(* CODESYS project Library.library
   Company: HDS Global
   Title: RoboFS_Standard
   Placeholder: RoboFS_Standard
   Version: 1.0

Project tree, tasks and I/O mapping:
  libraries: Tc2_MC2, * (Beckhoff Automation GmbH); Tc2_Standard, * (Beckhoff Automation GmbH); Tc2_System, * (Beckhoff Automation GmbH); Tc3_Module, * (Beckhoff Automation GmbH)
  Assemblies/
    function block Assembly_Conveyor [ST]
    function block Assembly_LAT [ST]
    function block Assembly_Lift [ST]
  Device Controllers/
    function block Device_Actuator [ST]
    function block Device_Motor_OnOff [ST]
    function block Device_PartSensor [FBD]
    function block Device_Servo [ST]: Disabled, Disabling, Enabled, Enabling, Error, Homing, Jogging, MoveComplete, MoveInProgress, Resetting, Stopped, Stopping
  DUTs/
    data type eInput
    data type Handshake_Receive
    data type Handshake_Send
    data type Intfc_Receiver
    data type Intfc_Sender
    data type ServoMove
  Enumerations/
    data type Cmd
    data type CmdActuator
    data type CmdMotorOnOff
    data type CmdServo
    data type Mode
    data type MoveTypeServo
    data type State
    data type StateActuator
    data type StateMotorOnOff
    data type StateSequencer
    data type StateServo
    data type StatusStep
  Instructions/
    function block eAND [ST]
    function block eOR [ST]
    function block MC_MoveParametersCheck [ST]
    function block StateManager [ST]
    function block Step [ST]
  Version/
    global variables Global_Version
*)

// DUTs/eInput
TYPE eInput :
STRUCT
	iState			: BOOL;
	iForceActive 	: BOOL;
	iForceInactive	: BOOL;
	cName			: STRING;
	cActiveState 	: BOOL := TRUE;
	oActive			: BOOL;
END_STRUCT
END_TYPE

// DUTs/Handshake_Receive
TYPE Handshake_Receive :
STRUCT
	ReadyToReceive 	: BOOL;
	Received		: BOOL;
	PartInfo		: STRING(20);
END_STRUCT
END_TYPE

// DUTs/Handshake_Send
TYPE Handshake_Send :
STRUCT
	WaitingToSend	: BOOL;
	Sending			: BOOL;
	PartInfo		: STRING(20);
END_STRUCT
END_TYPE

// DUTs/Intfc_Receiver
TYPE Intfc_Receiver :
STRUCT
	iHandshake 			: Handshake_Send;
	oHandshake			: Handshake_Receive;
	cSenderNetId		: STRING;
	cSenderPort			: UINT;
END_STRUCT
END_TYPE

// DUTs/Intfc_Sender
TYPE Intfc_Sender :
STRUCT
	oHandshake				: Handshake_Send;
	iHandshake		 		: Handshake_Receive;
	cReceiverNetId			: STRING;
	cReceiverPort			: UINT;
END_STRUCT
END_TYPE

// DUTs/ServoMove
TYPE ServoMove :
STRUCT
	Name 		: STRING;
	MoveType	: MoveTypeServo;
	Position	: LREAL;
	Velocity	: LREAL;
	Accel		: LREAL;
	Decel		: LREAL;
	Jerk		: LREAL;
	Direction	: MC_Direction;
	BufferMode	: MC_BufferMode;
	Permissive	: eAND;
	Interlock	: eAND;
END_STRUCT
END_TYPE

// Enumerations/Cmd
{attribute 'qualified_only'}
{attribute 'strict'}
TYPE Cmd :
(
	None,
	Abort,
	Reset,
	Start,
	Stop,
	Pause,
	Resume
);
END_TYPE

// Enumerations/CmdActuator
{attribute 'qualified_only'}
{attribute 'strict'}
TYPE CmdActuator :
(
	None,
	Extend,
	Retract,
	Reset
);
END_TYPE

// Enumerations/CmdMotorOnOff
{attribute 'qualified_only'}
{attribute 'strict'}
TYPE CmdMotorOnOff :
(
	None,
	Reset,
	StartFwd,
	StartRev,
	Stop	
);
END_TYPE

// Enumerations/CmdServo
{attribute 'qualified_only'}
{attribute 'strict'}
TYPE CmdServo :
(
	None,
	Enable,
	Disable,
	Reset,
	Home,
	StartMove,
	Stop,
	Jog
);
END_TYPE

// Enumerations/Mode
{attribute 'qualified_only'}
{attribute 'strict'}
TYPE Mode :
(
	Auto,
	Manual
);
END_TYPE

// Enumerations/MoveTypeServo
{attribute 'qualified_only'}
{attribute 'strict'}
TYPE MoveTypeServo :
(
	None,
	Continuous,
	LinearAbs,
	LinearRel,
	RotaryAbs,
	RotaryRel
);
END_TYPE

// Enumerations/State
{attribute 'qualified_only'}
{attribute 'strict'}
TYPE State :
(
	None,
	Stopped,
	Starting,
	Running,
	Pausing,
	Paused,
	Resuming,
	Stopping,
	Aborting,
	Aborted,
	Resetting	
);
END_TYPE

// Enumerations/StateActuator
{attribute 'qualified_only'}
{attribute 'strict'}
TYPE StateActuator :
(
	None,
	Error,
	Retracting,
	Retracted,
	Extending,
	Extended
);
END_TYPE

// Enumerations/StateMotorOnOff
{attribute 'qualified_only'}
{attribute 'strict'}
TYPE StateMotorOnOff :
(
	None,
	Error,
	Stopping,
	Stopped,
	StartingFwd,
	RunningFwd,
	StartingRev,
	RunningRev
);
END_TYPE

// Enumerations/StateSequencer
{attribute 'qualified_only'}
{attribute 'strict'}
TYPE StateSequencer :
(
	Idle,
	Running,
	Complete,
	Faulted
);
END_TYPE

// Enumerations/StateServo
{attribute 'qualified_only'}
{attribute 'strict'}
TYPE StateServo :
(
	None,
	Error,
	Resetting,
	Disabling,
	Disabled,
	Enabling,
	Enabled,
	Homing,
	MoveInProgress,
	MoveComplete,
	Stopping,	
	Stopped,
	Jogging
);
END_TYPE

// Enumerations/StatusStep
{attribute 'qualified_only'}
{attribute 'strict'}
TYPE StatusStep :
(
	Inactive,
	Active,
	Faulted,
	TimedOut,
	Complete
);
END_TYPE

// Version/Global_Version
{attribute 'TcGenerated'}
// This function has been automatically generated from the project information.
VAR_GLOBAL CONSTANT
	{attribute 'const_non_replaced'}
	{attribute 'linkalways'}
	stLibVersion_RoboFS_Standard : ST_LibVersion := (iMajor := 1, iMinor := 0, iBuild := 0, iRevision := 0, sVersion := '1.0');
END_VAR

// Assemblies/Assembly_Conveyor
FUNCTION_BLOCK Assembly_Conveyor
VAR_INPUT
	cmdRunFwd 			: BOOL;
	cmdRunRev 			: BOOL;
	cmdStop 			: BOOL;
	cfgRestartDelay		: TIME;
	inpTensionOK AT %I*	: BOOL;
END_VAR
VAR_OUTPUT
END_VAR
VAR
END_VAR

END_FUNCTION_BLOCK

// Assemblies/Assembly_LAT
FUNCTION_BLOCK Assembly_LAT

VAR_INPUT
	iSafetyOK			: BOOL := TRUE;
	iPowerOn			: BOOL;
	cmdDivertRight 		: BOOL;
	cmdDivertLeft 		: BOOL;
	cmdPassThru 		: BOOL;
	cmdReceiveRight 	: BOOL;
	cmdReceiveLeft 		: BOOL;
END_VAR

VAR_OUTPUT
	stsIdle				: BOOL;
	stsDivertingRight 	: BOOL;
	stsDivertingLeft 	: BOOL;
	stsPassingThru 		: BOOL;
	stsReceivingRight	: BOOL;
	stsRecevingLeft 	: BOOL;
	stsFaulted 			: BOOL;
	stsFaultCode 		: INT;
END_VAR

VAR_IN_OUT
	PartSensor 			: Device_PartSensor;
	Lift 				: Device_Actuator;
	Transfer			: Device_Motor_OnOff;
END_VAR

VAR
END_VAR

//Map SafetyOK input to Lift and Conv

Lift.iSafetyOK 	:= inpSafetyOK;
Conv.inpSafetyOK 	:= inpSafetyOK;

//Map PowerOn input to Lift and Conv

Lift.iPowerOn 	:= inpPowerOn;
Conv.inpPowerOn 	:= inpPowerOn;

IF PartSensor.oPartPresent THEN
	//Lift.cmdExtend 	:= 1;
	//Conv.cmdRunFwd 	:= 1;
END_IF

END_FUNCTION_BLOCK

// Device Controllers/Device_PartSensor
FUNCTION_BLOCK Device_PartSensor

VAR_INPUT
	iSensor1On AT %I* 	: BOOL;
END_VAR

VAR_OUTPUT
	oPartPresent		: BOOL;
END_VAR

VAR_INPUT PERSISTENT
	Name				: STRING;
	
	cOnDelay 			: TIME;
	cOffDelay 			: TIME;
END_VAR

VAR
	OnDelayTimer 		: TON;
	OffDelayTimer 		: TOF;
	SetReset: SR;
END_VAR

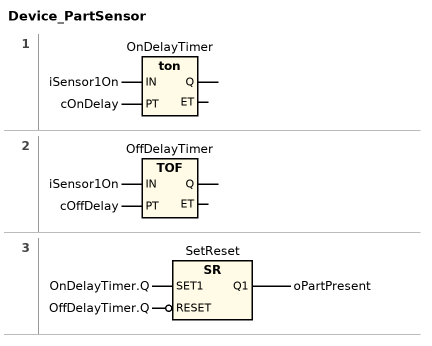
// NETWORK 1
OnDelayTimer(IN := iSensor1On, PT := cOnDelay); // ton

// NETWORK 2
OffDelayTimer(IN := iSensor1On, PT := cOffDelay); // TOF

// NETWORK 3
SetReset(SET1 := OnDelayTimer.Q, RESET := NOT OffDelayTimer.Q); // SR
oPartPresent := SetReset.Q1;

END_FUNCTION_BLOCK

// Device Controllers/Device_Actuator
FUNCTION_BLOCK Device_Actuator

VAR_INPUT
	iPowerOn 			: BOOL;
	iSafetyOK 			: BOOL;
	iMode				: Mode;
	iCmd 				: CmdActuator;
	iCmdRetry			: BOOL;
	iCmdAbort			: BOOL;
	iOkToExtend			: eAND;
	iOkToRetract		: eAND;

	iExtended AT %I* 	: BOOL;
	iRetracted AT %I* 	: BOOL;
END_VAR

VAR_OUTPUT
	oState				: StateActuator;
	oErrorCode			: INT;
	oCmdFailed			: BOOL;	
	
	oExtend AT %Q* 		: BOOL;
	oRetract AT %Q* 	: BOOL;
END_VAR

VAR
	ExtendedDebounce	: TON;
	ExtendingTimer		: TON;
	RetractedDebounce	: TON;
	RetractingTimer		: TON;
END_VAR

VAR_INPUT PERSISTENT	
	Name				: STRING;
	ExtendAlias			: STRING;
	RetractAlias		: STRING;

	cHold 				: BOOL 	:= 1;
	cDebounceTime		: TIME	:= T#0.5S;
	cExtendTimeout 		: TIME	:= T#5S;
	cRetractTimeout 	: TIME	:= T#5S;	
END_VAR

ExtendedDebounce.PT := cDebounceTime;
RetractedDebounce.PT := cDebounceTime;
ExtendingTimer.PT := cExtendTimeout;
RetractingTimer.PT := cRetractTimeout;

ExtendedDebounce (IN :=iExtended);
RetractedDebounce (IN := iRetracted);


CASE oState OF
//0=============================================================================================================//
	StateActuator.None:
								IF iCmd = CmdActuator.Retract THEN
									IF iOkToRetract.Q AND NOT oCmdFailed THEN
										oState 			:= StateActuator.Retracting;
										iCmd			:= CmdActuator.None;
									ELSE
										oCmdFailed 		:= TRUE;
										IF iCmdRetry THEN
											oCmdFailed	:= FALSE;
											iCmdRetry	:= FALSE;
										ELSIF iCmdAbort THEN
											oCmdFailed	:= FALSE;
											iCmdAbort	:= FALSE;
											iCmd		:= CmdActuator.None;
										END_IF
									END_IF
								ELSIF iCmd = CmdActuator.Extend THEN
									IF iOkToExtend.Q AND NOT oCmdFailed THEN
									oState 				:= StateActuator.Extending;
									iCmd				:= CmdActuator.None;
									ELSE
										oCmdFailed 		:= TRUE;
										IF iCmdRetry THEN
											oCmdFailed	:= FALSE;
											iCmdRetry	:= FALSE;
										ELSIF iCmdAbort THEN
											oCmdFailed	:= FALSE;
											iCmdAbort	:= FALSE;
											iCmd		:= CmdActuator.None;
										END_IF
									END_IF
								END_IF
//1=============================================================================================================//	
	StateActuator.Error:
								IF iCmd = CmdActuator.Reset THEN
									IF ExtendedDebounce.Q THEN
										oState 		:= StateActuator.Extended;
										oExtend 	:= cHold;
										oRetract 	:= FALSE;
									ELSIF RetractedDebounce.Q THEN
										oState 		:= StateActuator.Retracted;
										oExtend		:= FALSE;
										oRetract 	:= cHold;
									ELSE
										oState 		:= StateActuator.None;
										oExtend 	:= FALSE;
										oRetract 	:= FALSE;
									END_IF
								END_IF
								IF oState <> StateActuator.Error THEN
									oErrorCode 		:= 0;
								END_IF
//2=============================================================================================================//	
	StateActuator.Extending:
								oExtend 		:= TRUE;
								oRetract		:= FALSE;
								
								IF ExtendedDebounce.Q THEN
									oState := StateActuator.Extended;
									oExtend := cHold;
								ELSE
									ExtendingTimer (IN := TRUE);
									IF ExtendingTimer.Q THEN
										oState := StateActuator.Error;
										oErrorCode := 1;														//	Failed to Extend
									END_IF
								END_IF
														
								IF oState <> StateActuator.Extending THEN
									ExtendingTimer (IN := FALSE);
								END_IF
//3=============================================================================================================//
	StateActuator.Extended:
								IF cHold AND NOT iExtended THEN
									oState:= StateActuator.Error;
									oErrorcode := 2;															//	Failed to remain Extended
								END_IF
								
								IF iCmd = CmdActuator.Retract THEN
									IF iOkToRetract.Q AND NOT oCmdFailed THEN
										oState 			:= StateActuator.Retracting;
										iCmd			:= CmdActuator.None;
									ELSE
										oCmdFailed 		:= TRUE;
										IF iCmdRetry THEN
											oCmdFailed	:= FALSE;
											iCmdRetry	:= FALSE;
										ELSIF iCmdAbort THEN
											oCmdFailed	:= FALSE;
											iCmdAbort	:= FALSE;
											iCmd		:= CmdActuator.None;
										END_IF
									END_IF
								END_IF
//4=============================================================================================================//	
	StateActuator.Retracting:
								oRetract 		:= TRUE;
								oExtend			:= FALSE;
								
								IF RetractedDebounce.Q THEN
									oState := StateActuator.Retracted;
									oRetract := cHold;
								ELSE
									RetractingTimer (IN := TRUE);
									IF RetractingTimer.Q THEN
										oState := StateActuator.Error;
										oErrorCode := 3;														//	Failed to Retract
									END_IF
								END_IF
								
								IF oState <> StateActuator.Retracting THEN
									RetractingTimer (IN := FALSE);
								END_IF
//5=============================================================================================================//								
	StateActuator.Retracted:
								IF cHold AND NOT iRetracted THEN
									oState:= StateActuator.Error;
									oErrorcode := 4;															//	Failed to remain Retracted
								END_IF
								
								IF iCmd = CmdActuator.Extend THEN
									IF iOkToExtend.Q AND NOT oCmdFailed THEN
									oState 				:= StateActuator.Extending;
									iCmd				:= CmdActuator.None;
									ELSE
										oCmdFailed 		:= TRUE;
										IF iCmdRetry THEN
											oCmdFailed	:= FALSE;
											iCmdRetry	:= FALSE;
										ELSIF iCmdAbort THEN
											oCmdFailed	:= FALSE;
											iCmdAbort	:= FALSE;
											iCmd		:= CmdActuator.None;
										END_IF
									END_IF
								END_IF
END_CASE

END_FUNCTION_BLOCK

// Instructions/eAND
FUNCTION_BLOCK eAND
VAR_INPUT
	IN1 : BOOL;
	IN2 : BOOL;
	IN3 : BOOL;
	IN4 : BOOL;
	IN5 : BOOL;
	IN6	: BOOL;
	IN7	: BOOL;
	IN8 : BOOL;
	IN9	: BOOL;
	IN10 : BOOL;
	
	Initialize : BOOL := TRUE;
END_VAR

VAR_OUTPUT
	Q : BOOL;
END_VAR

VAR
	Input : ARRAY [1..10] OF eInput;
	n : INT;
END_VAR

IF Initialize THEN
	IN1 := Input[1].cActiveState;
	IN2 := Input[2].cActiveState;
	IN3 := Input[3].cActiveState;
	IN4 := Input[4].cActiveState;
	IN5 := Input[5].cActiveState;
	IN6 := Input[6].cActiveState;
	IN7 := Input[7].cActiveState;
	IN8 := Input[8].cActiveState;
	IN9 := Input[9].cActiveState;
	IN10 := Input[10].cActiveState;	
END_IF

Input[1].iState := IN1;
Input[2].iState := IN2;
Input[3].iState := IN3;
Input[4].iState := IN4;
Input[5].iState := IN5;
Input[6].iState := IN6;
Input[7].iState := IN7;
Input[8].iState := IN8;
Input[9].iState := IN9;
Input[10].iState := IN10;


FOR n := 1 TO 10 BY 1 DO

		IF Input[n].iForceActive AND NOT Input[n].iForceInactive THEN
			Input[n].oActive := TRUE;
		ELSIF Input[n].iForceInactive AND NOT Input[n].iForceActive THEN
			Input[n].oActive := FALSE;
		ELSIF Input[n].cActiveState = Input[n].iState THEN
			Input[n].oActive := TRUE;
		ELSIF Input[n].cActiveState <> Input[n].iState THEN
			Input[n].oActive := FALSE;
		END_IF

END_FOR	

IF NOT Initialize THEN
Q := 	Input[1].oActive AND 
		Input[2].oActive AND 
		Input[3].oActive AND 
		Input[4].oActive AND 
		Input[5].oActive AND 
		Input[6].oActive AND 
		Input[7].oActive AND 
		Input[8].oActive AND 
		Input[9].oActive AND 
		Input[10].oActive;
END_IF

Initialize := FALSE;

END_FUNCTION_BLOCK

// Device Controllers/Device_Motor_OnOff
FUNCTION_BLOCK Device_Motor_OnOff
VAR_INPUT
	iPowerOn 		: BOOL;
	iSafetyOK 		: BOOL;
	iCmd 			: CmdMotorOnOff;
	iCmdRetry		: BOOL;
	iCmdAbort		: BOOL;
	iOkToRunFwd		: eAND;
	iOkToRunRev		: eAND;

	iFwdOn AT %I* 	: BOOL;
	iRevOn AT %I* 	: BOOL;
END_VAR

VAR_OUTPUT
	oState			: StateMotorOnOff;
	oCmdFailed		: BOOL;
	oErrorCode		: INT;
	
	oRunFwd AT %Q* 	: BOOL;
	oRunRev AT %Q* 	: BOOL;
END_VAR

VAR_INPUT PERSISTENT
	Name			: STRING;
	
	cReversible 	: BOOL;
	cStartTimeout 	: TIME := T#5S;
	cStopTimeout 	: TIME := T#5S;
END_VAR

VAR
	StartTimer		: TON;
	StopTimer		: TON;
END_VAR

StartTimer.PT 	:= cStartTimeout;
StopTimer.PT 	:= cStopTimeout;

CASE oState OF
//0=============================================================================================================//
	StateMotorOnOff.None:
								oState 				:= StateMotorOnOff.Stopping;
//1=============================================================================================================//									
	StateMotorOnOff.Error:
								IF iCmd = CmdMotorOnOff.Reset THEN
									oState 			:= StateMotorOnOff.Stopping;
									iCmd			:= CmdMotorOnOff.None;	
								END_IF
//2=============================================================================================================//	
	StateMotorOnOff.Stopping:
								oRunFwd 			:= FALSE;
								oRunRev 			:= FALSE;
								IF NOT iFwdOn AND NOT iRevOn THEN
									oState 			:= StateMotorOnOff.Stopped;
								ELSE
									StopTimer(IN 	:= TRUE);
									IF StopTimer.Q THEN
										oState 		:= StateMotorOnOff.Error;
										oErrorCode 	:= 5;														//	Failed to Stop
									END_IF
								END_IF
								
								IF oState <> StateMotorOnOff.Stopping THEN
									StopTimer(IN 	:= FALSE);
								END_IF
//3=============================================================================================================//								
	StateMotorOnOff.Stopped:
								CASE iCmd OF
									CmdMotorOnOff.StartFwd:
										IF iOkToRunFwd AND NOT oCmdFailed THEN
											oState		:= StateMotorOnOff.StartingFwd;
											iCmd 		:= CmdMotorOnOff.None;
										ELSE
											oCmdFailed 	:= TRUE;
											IF iCmdRetry THEN
												oCmdFailed	:= FALSE;
												iCmdRetry	:= FALSE;
											ELSIF iCmdAbort THEN
												oCmdFailed	:= FALSE;
												iCmdAbort	:= FALSE;
												iCmd		:= CmdMotorOnOff.None;
											END_IF
										END_IF
										
									CmdMotorOnOff.StartRev:
										IF iOkToRunRev AND cReversible AND NOT oCmdFailed THEN
											oState		:= StateMotorOnOff.StartingFwd;
											iCmd 		:= CmdMotorOnOff.None;
										ELSE
											oCmdFailed 	:= TRUE;
											IF iCmdRetry THEN
												oCmdFailed	:= FALSE;
												iCmdRetry	:= FALSE;
											ELSIF iCmdAbort THEN
												oCmdFailed	:= FALSE;
												iCmdAbort	:= FALSE;
												iCmd		:= CmdMotorOnOff.None;
											END_IF
										END_IF
								END_CASE
//4=============================================================================================================//								
	StateMotorOnOff.StartingFwd:
								oRunFwd 			:= TRUE;
								oRunRev 			:= FALSE;
								IF iFwdOn AND NOT iRevOn THEN
									oState := StateMotorOnOff.RunningFwd;
								ELSE
									StartTimer(IN 	:= TRUE);
									IF StartTimer.Q THEN
										oState 		:= StateMotorOnOff.Error;	
										oErrorCode 	:= 1;														//	Failed to Start Fwd
									END_IF	
								END_IF
								
								CASE iCmd OF
									CmdMotorOnOff.Stop:
										oState		:= StateMotorOnOff.Stopping;
										iCmd		:= CmdMotorOnOff.None;
								END_CASE
								
								IF oState <> StateMotorOnOff.StartingFwd THEN
									StartTimer(IN 	:= FALSE);
								END_IF
								
//5=============================================================================================================//								
	StateMotorOnOff.RunningFwd:
								IF NOT iFwdOn OR iRevOn THEN
									oState			:= StateMotorOnOff.Error;
									oErrorCode		:= 2;														//	Failed to Remain Running Fwd
								END_IF
								
								CASE iCmd OF
									CmdMotorOnOff.Stop:
										oState		:= StateMotorOnOff.Stopping;
										iCmd		:= CmdMotorOnOff.None;
								END_CASE
//6=============================================================================================================//	
	StateMotorOnOff.StartingRev:
								oRunFwd 			:= FALSE;
								oRunRev 			:= TRUE;
								
								IF iFwdOn AND NOT iRevOn THEN
									oState 			:= StateMotorOnOff.RunningFwd;
								ELSE
									StartTimer(IN 	:= TRUE);
									IF StartTimer.Q THEN
										oState 		:= StateMotorOnOff.Error;
										oErrorCode 	:= 3;														//	Failed to Start Rev
									END_IF
								END_IF
								
								IF oState <> StateMotorOnOff.StartingFwd THEN
									StartTimer(IN 	:= FALSE);
								END_IF
//7=============================================================================================================//								
	StateMotorOnOff.RunningRev:
								IF NOT iRevOn OR iFwdOn THEN
									oState			:= StateMotorOnOff.Error;
									oErrorCode		:= 4;														//	Failed to Remain Running Rev
								END_IF
								
								CASE iCmd OF
									CmdMotorOnOff.Stop:
										oState		:= StateMotorOnOff.Stopping;
										iCmd		:= CmdMotorOnOff.None;
								END_CASE
	
END_CASE

END_FUNCTION_BLOCK

// Assemblies/Assembly_Lift
FUNCTION_BLOCK Assembly_Lift

VAR_INPUT
	iPowerOn			: BOOL;
	iSafetyOk			: BOOL;
	cmdRaise			: BOOL;
	cmdLower			: BOOL;
	cfgReverseAction	: BOOL;
END_VAR

VAR_OUTPUT
	stsRaised			: BOOL;
	stsLowered			: BOOL;
	stsFaulted			: BOOL;
	stsFaultCode		: BOOL;
END_VAR

VAR_IN_OUT
	Actuator : Device_Actuator;
END_VAR

END_FUNCTION_BLOCK

// Device Controllers/Device_Servo
FUNCTION_BLOCK Device_Servo

VAR_INPUT
	iPowerOn				: BOOL;							//	Power On signal
	iSafetyOk				: BOOL;							//	Safety Ok signal from safety logic
	iMode					: Mode;							// 	Device Mode - Auto/Manual
	iCmd					: CmdServo;						// 	Servo command
	iCmdRetry				: BOOL;							// 	Retry current Command (when failed)
	iCmdAbort				: BOOL;							// 	Abort current Command (when failed)
	iMoveIndex				: INT;							// 	Servo Move Index (command)
	iJogFwd					: BOOL;							// 	Jog Forward command
	iJogRev					: BOOL;							// 	Jog Reverse command
	iJogFast				: BOOL;							// 	Jog at standard fast speed
END_VAR

VAR_OUTPUT
	oState					: StateServo := StateServo.Disabled;	// Servo Status
	oErrorCode				: INT;
	oCmdFailed				: BOOL;									// Current Command failed to execute
	sMoveIndex				: INT;									// Servo Move Index (status)
	sMoveNotPermitted		: BOOL;									// Specified move permissives are not active
	sMoveInvalid			: BOOL;									// Specified move does not have valid parameters
END_VAR

VAR_IN_OUT
	ioAxis					: AXIS_REF;						// Axis reference (process data plc/nc)	
	ioMoves					: ARRAY[1..100] OF ServoMove; 	// Array of Servo Moves
END_VAR

VAR	
	MCPower 				: MC_Power;						// FB for enable and override
	MCReset 				: MC_Reset;						// FB to reset axis
	MCHome					: MC_Home;						// FB to home axis
	MCHalt	 				: MC_Halt;						// FB to stop axis
	MCMoveVel				: MC_MoveVelocity;				// FB for continuous velocity moves
	MCMoveAbs				: MC_MoveAbsolute;				// FB for absolute position moves
	MCMoveRel				: MC_MoveRelative;				// FB for relative position moves
	MCJog					: MC_Jog;						// FB for jogging
	MCMoveParametersCheck	: MC_MoveParametersCheck;		// FB for validating move parameters
	JogMode					: E_JogMode;					// ENUM for jog mode
	CurrentMove				: ServoMove;
END_VAR

VAR PERSISTENT
	Name					: STRING;
END_VAR

VAR_TEMP
	MoveIsValid		: BOOL;
	PrevStatus		: StateServo;
END_VAR

ioAxis.ReadStatus();

CASE oState OF
	StateServo.None:			oState := StateServo.Disabling;
	StateServo.Error:			Error();	
	StateServo.Resetting:		Resetting();
	StateServo.Disabling:		Disabling();
	StateServo.Disabled:		Disabled();
	StateServo.Enabling:		Enabling();
	StateServo.Enabled:			Enabled();
	StateServo.Homing:			Homing();
	StateServo.MoveInProgress:	MoveInProgress();																				//	CurrentMove is set in the previous state
	StateServo.MoveComplete :	MoveComplete();
	StateServo.Stopping:		Stopping();
	StateServo.Stopped:			Stopped();
	StateServo.Jogging :		Jogging();
END_CASE

ACTION Disabled:
IF 	iCmd = CmdServo.Enable THEN												//	accept the Enable command
	oState 					:= StateServo.Enabling;							//	change status to Enabling
	iCmd 					:= CmdServo.None;								//	clear command
END_IF

IF ioAxis.Status.Error THEN
	oState						:= StateServo.Error;
ELSIF ioAxis.Status.StandStill THEN
	oState						:= StateServo.Enabled;
END_IF
END_ACTION

ACTION Disabling:
MCPower(	Enable 				:= FALSE,										//	call fb to Disable axis
			Enable_Positive		:= FALSE, 										//
			Enable_Negative		:= FALSE, 										//
			Override			:= 0,											//
			Axis				:= ioAxis);										//
IF 	NOT MCPower.Status AND ioAxis.Status.Disabled THEN							//	check whether fb is Done and axis status is Disabled
	oState 						:= StateServo.Disabled;								//	change status to Disabled
END_IF

IF MCPower.Error THEN
	oCmdFailed					:= TRUE;
	IF iCmdRetry THEN
		MCPower( 	Enable		:= TRUE,										//	call Power fb with Enable = true
					Axis		:= ioAxis);										//	Power fb will get retriggered on the next scan
		oCmdFailed				:= FALSE;
		iCmdRetry				:= FALSE;
	ELSIF iCmdAbort THEN
		MCPower( 	Enable		:= TRUE,										//	call Power fb with Enable = true
					Axis		:= ioAxis);
		oState					:= PrevStatus;									//	change status back to previous
		oCmdFailed				:= FALSE;
		iCmdAbort				:= FALSE;
	END_IF
END_IF

IF ioAxis.Status.Error THEN
	oState						:= StateServo.Error;
END_IF
END_ACTION

ACTION Enabled:
IF ioAxis.Status.Homed THEN														//	check whether the axis has been homed
	oState 					:= StateServo.Stopped;								//	change status to Stopped
ELSIF ioAxis.Status.Error THEN													//	check whether the axis is in error
	oState						:= StateServo.Error;							//	change status to Error
END_IF

CASE iCmd  OF
		CmdServo.Home:															//	accept the Home command
					oState		:= StateServo.Homing;							//	change status to Homing
					iCmd	:= CmdServo.None;								//	clear command
		CmdServo.Jog:															//	accept the Jog Command
					oState		:= StateServo.Jogging;							//	change status to Jogging
					iCmd	:= CmdServo.None;								//	clear command
		CmdServo.Disable:														//	accept the Disable command
					oState		:= StateServo.Disabling;						//	change status to Disabling
					PrevStatus	:= StateServo.Enabled;
					iCmd	:= CmdServo.None;								//	clear command  
END_CASE
END_ACTION

ACTION Enabling:
MCPower(	Enable 				:= TRUE, 										//	call fb to Enable axis
			Enable_Positive		:= TRUE, 										//					
			Enable_Negative		:= TRUE, 										//
			Override			:= 100,											//
			Axis				:= ioAxis);										//
IF 	MCPower.Status AND ioAxis.Status.StandStill THEN							//	check whether fb is Done and axis status is Standstill
	oState 					:= StateServo.Enabled;								//	change status to Enabled 
END_IF

IF MCPower.Error THEN
	oCmdFailed				:= TRUE;
	IF iCmdRetry THEN
		MCPower( 	Enable		:= FALSE,										//	call Power fb with Execute = false
					Axis		:= ioAxis);										//	Power fb will get retriggered on the next scan
		oCmdFailed			:= FALSE;
		iCmdRetry			:= FALSE;
	ELSIF iCmdAbort THEN
		MCPower( 	Enable		:= FALSE,										//	call Power fb with Execute = false
					Axis		:= ioAxis);
		oState					:= StateServo.Disabled;
		oCmdFailed			:= FALSE;
		iCmdAbort			:= FALSE;
	END_IF
END_IF

IF ioAxis.Status.Error THEN
	oState						:= StateServo.Error;
END_IF
END_ACTION

ACTION Error:
IF 	iCmd = CmdServo.Reset THEN												//	accept the Reset command
	oState		 				:= StateServo.Resetting;							//	change status to Resetting		
	iCmd 						:= CmdServo.None;								//	clear command
END_IF								
																				//	(for error reset externally, for ex. by power cycle of drive)
IF ioAxis.Status.Disabled AND NOT ioaxis.status.error THEN						//	check whether axis status is Disabled
	oState						:= StateServo.Disabled;							//	change status to Disabled
ELSIF ioAxis.Status.StandStill THEN												//	or else if axis status is Standstill	
	oState						:= StateServo.Enabled;							//	change status to Enabled
END_IF
END_ACTION

ACTION Homing:
MCHome( 	Execute				:= TRUE,										//	call fb to Home axis
			Axis				:= ioAxis);
IF 	MCHome.Done THEN 
	IF ioAxis.Status.Homed AND ioAxis.Status.StandStill THEN					//	check for fb Done and axis status successfully changed to Homed and Standstill
	oState 					:= StateServo.Stopped;							//	change status to Stopped
	END_IF
ELSIF MCHome.Error THEN
	oCmdFailed				:= TRUE;
	IF iCmdRetry THEN														//	command retry
		MCHome( 	Execute		:= FALSE,										//	call Home fb with Execute = false
					Axis		:= ioAxis);										//	Home fb will get retriggered on the next scan
		oCmdFailed			:= FALSE;
		iCmdRetry			:= FALSE;
	ELSIF iCmdAbort THEN													//	command abort
		oState					:= StateServo.Enabled;								//	change status back to Error
		oCmdFailed			:= FALSE;
		iCmdAbort			:= FALSE;
	END_IF
END_IF

IF 	iCmd = CmdServo.Stop THEN												//	accept the Stop command
	oState 					:= StateServo.Stopping;							//	change status to Stopping
ELSIF iCmd = CmdServo.Disable THEN												//	accept the Disable command
	oState 					:= StateServo.Disabling;							//	change status to Disabling
END_IF

IF ioAxis.Status.Error THEN
	oState						:= StateServo.Error;
END_IF

IF oState <> StateServo.Homing THEN												//	when Status has been changed within the block
	MCHome( Execute				:= FALSE,										//	call Home fb with Execute = false
			Axis				:= ioAxis);
	iCmd 					:= CmdServo.None;								//	clear command
END_IF
END_ACTION

ACTION Jogging:
IF iJogFast THEN																//	check whether JogFast is true
	JogMode							:= E_JogMode.MC_JOGMODE_STANDARD_FAST;		//	set fast jog mode
ELSE																			//
	JogMode							:= E_JogMode.MC_JOGMODE_STANDARD_SLOW;		//	default jog mode is slow
END_IF																			//
																				//
MCJog(		JogForward				:= iJogFwd,									//	call fb for Jogging
			JogBackwards			:= iJogRev, 								//	(exclusivity of JogFwd and JogRev must be enforced at the input source)
			Mode					:= JogMode,									//
			Axis					:= ioAxis);									//
																				//
IF NOT MCJog.Busy THEN															//	when tmpfbStatus=True this indicates no jog in progress
	CASE iCmd OF																//
		CmdServo.StartMove:														//	accept the StartMove command
			ioMoves[iMoveIndex].Permissive();									//	check permissive
			IF NOT ioMoves[iMoveIndex].Permissive.Q THEN
				sMoveNotPermitted				:= TRUE;
				oCmdFailed						:= TRUE;
			ELSE
				sMoveNotPermitted				:= FALSE;
			END_IF
			
			MCMoveParametersCheck(	iMoveIndex 	:= iMoveIndex,					//	check parameters
									ioMoves 	:= ioMoves, 
									ioAxis 		:= ioAxis);
			IF NOT MCMoveParametersCheck.oValid THEN
				sMoveInvalid					:= TRUE;
				oCmdFailed						:= TRUE;
			ELSE
				sMoveInvalid					:= FALSE;
			END_IF
					
			IF  ioMoves[iMoveIndex].Permissive.Q AND MCMoveParametersCheck.oValid AND NOT oCmdFailed THEN
				CurrentMove 			:= ioMoves[iMoveIndex];
				oState 					:= StateServo.MoveInProgress;
				iCmd 					:= CmdServo.None;						//	clear command
			END_IF
			
			IF oCmdFailed AND iCmdRetry THEN
				oCmdFailed				:= FALSE;
				iCmdRetry				:= FALSE;
			ELSIF oCmdFailed AND iCmdAbort THEN
				oCmdFailed				:= FALSE;	 	
				sMoveNotPermitted		:= FALSE;
				sMoveInvalid			:= FALSE;	
				iCmd	 				:= CmdServo.None;						//	clear command
				iCmdAbort				:= FALSE;
			END_IF	
		CmdServo.Stop:															//	accept Stop command		
			oState 					:= StateServo.Stopping;						//	change status to Stopping
			PrevStatus				:= StateServo.Jogging;
			iCmd 					:= CmdServo.None;							//	clear command
			iJogFast				:= FALSE;									//	clear fast mode for jogging
		CmdServo.Disable:														//	accept Disable command
			oState 					:= StateServo.Disabling;					//	change status to Disabling
			iCmd 					:= CmdServo.None;							//	clear command
			iJogFast				:= FALSE;									//	clear fast mode for jogging
	END_CASE
END_IF

IF ioAxis.Status.Error THEN
	oState						:= StateServo.Error;
END_IF
END_ACTION

ACTION MoveComplete:
CASE iCmd OF
	CmdServo.Disable:
		oState 						:= StateServo.Disabling;
		iCmd 						:= CmdServo.None;								//	clear command
	CmdServo.Stop:
		oState 						:= StateServo.Stopping;
		PrevStatus					:= StateServo.MoveComplete;
		iCmd 						:= CmdServo.None;								//	clear command
	CmdServo.StartMove:
		ioMoves[iMoveIndex].Permissive();										//	check permissive
		IF NOT ioMoves[iMoveIndex].Permissive.Q THEN
			sMoveNotPermitted				:= TRUE;
			oCmdFailed						:= TRUE;
		ELSE
			sMoveNotPermitted				:= FALSE;
		END_IF
		
		MCMoveParametersCheck(	iMoveIndex 	:= iMoveIndex,						//	check parameters
								ioMoves 	:= ioMoves, 
								ioAxis 		:= ioAxis);
		IF NOT MCMoveParametersCheck.oValid THEN
			sMoveInvalid					:= TRUE;
			oCmdFailed						:= TRUE;
		ELSE
			sMoveInvalid					:= FALSE;
		END_IF
				
		IF  ioMoves[iMoveIndex].Permissive.Q AND MCMoveParametersCheck.oValid AND NOT oCmdFailed THEN
			CurrentMove 			:= ioMoves[iMoveIndex];
			oState 					:= StateServo.MoveInProgress;
			iCmd 					:= CmdServo.None;							//	clear command
		END_IF
		
		IF oCmdFailed AND iCmdRetry THEN
			oCmdFailed				:= FALSE;
			iCmdRetry				:= FALSE;
		ELSIF oCmdFailed AND iCmdAbort THEN
			oCmdFailed				:= FALSE;
			sMoveNotPermitted		:= FALSE;
			sMoveInvalid			:= FALSE;		 		
			iCmd	 				:= CmdServo.None;							//	clear command
			iCmdAbort				:= FALSE;
		END_IF		
	CmdServo.Jog:
		oState 					:= StateServo.Jogging;
		iCmd 					:= CmdServo.None;								//	clear command
END_CASE

IF ioAxis.Status.Error THEN
	oState						:= StateServo.Error;
END_IF
END_ACTION

ACTION MoveInProgress:
CASE CurrentMove.MoveType OF
 
	MoveTypeServo.Continuous :
				MCMoveVel (	Execute 		:= TRUE,
							Velocity		:= CurrentMove.Velocity,
							Acceleration	:= CurrentMove.Accel,
							Deceleration	:= CurrentMove.Decel,
							Jerk			:= CurrentMove.Jerk,
							BufferMode		:= CurrentMove.BufferMode,
							Direction		:= CurrentMove.Direction,
							Axis 			:= ioAxis);
				IF MCMoveVel.InVelocity THEN
					oState					:= StateServo.MoveComplete;
				ELSIF MCMoveVel.Error THEN
					oCmdFailed			:= TRUE;
					IF iCmdRetry THEN										//	command retry
						MCMoveVel( 	Execute	:= FALSE,							//	call Move fb with Execute = false
									Axis	:= ioAxis);							//	Home fb will get retriggered on the next scan
						oCmdFailed		:= FALSE;
						iCmdRetry		:= FALSE;
					ELSIF iCmdAbort THEN									//	command abort
						oState				:= StateServo.Stopping;				//	change status to Stopping
						oCmdFailed		:= FALSE;
						iCmdAbort		:= FALSE;
					END_IF
				END_IF
							
	MoveTypeServo.LinearAbs :
				MCMoveAbs (	Execute 		:= TRUE,
							Position		:= CurrentMove.Position,
							Velocity		:= CurrentMove.Velocity,
							Acceleration	:= CurrentMove.Accel,
							Deceleration	:= CurrentMove.Decel,
							Jerk			:= CurrentMove.Jerk,
							BufferMode		:= CurrentMove.BufferMode,
							Axis 			:= ioAxis);
				IF MCMoveAbs.Done THEN
					oState					:= StateServo.MoveComplete;
				ELSIF MCMoveAbs.Error THEN
					oCmdFailed			:= TRUE;
					IF iCmdRetry THEN										//	command retry
						MCMoveAbs( 	Execute	:= FALSE,							//	call Move fb with Execute = false
									Axis	:= ioAxis);							//	Move fb will get retriggered on the next scan
						oCmdFailed		:= FALSE;
						iCmdRetry		:= FALSE;
					ELSIF iCmdAbort THEN									//	command abort
						oState				:= StateServo.Stopping;				//	change status to Stopping
						oCmdFailed		:= FALSE;
						iCmdAbort		:= FALSE;
					END_IF
				END_IF
				
	MoveTypeServo.LinearRel :
				MCMoveRel (	Execute 		:= TRUE,
							Distance		:= CurrentMove.Position,			// Current Move Position is expected to be 'distance' for this move type
							Velocity		:= CurrentMove.Velocity,
							Acceleration	:= CurrentMove.Accel,
							Deceleration	:= CurrentMove.Decel,
							Jerk			:= CurrentMove.Jerk,
							BufferMode		:= CurrentMove.BufferMode,
							Axis 			:= ioAxis);
				IF MCMoveRel.Done THEN
					oState					:= StateServo.MoveComplete;
				ELSIF MCMoveRel.Error THEN
					oCmdFailed			:= TRUE;
					IF iCmdRetry THEN										//	command retry
						MCMoveRel( 	Execute	:= FALSE,							//	call Move fb with Execute = false
									Axis	:= ioAxis);							//	Move fb will get retriggered on the next scan
						oCmdFailed		:= FALSE;
						iCmdRetry		:= FALSE;
					ELSIF iCmdAbort THEN									//	command abort
						oState			:= StateServo.Stopping;				//	change status to Stopping
						oCmdFailed		:= FALSE;
						iCmdAbort		:= FALSE;
					END_IF
				END_IF
				
	MoveTypeServo.RotaryAbs :
	MoveTypeServo.RotaryRel :
END_CASE
	
CASE iCmd OF
	CmdServo.Disable:															//	accept the Disable command
		oState 					:= StateServo.Disabling;						//	change status to Disabling
	CmdServo.Stop:																//	accept the Stop command
		oState 					:= StateServo.Stopping;						//	chagne status to Stopping
		PrevStatus					:= StateServo.MoveInProgress;
END_CASE
	
IF ioAxis.Status.Error THEN
	oState							:= StateServo.Error;
END_IF
	
IF oState <> StateServo.MoveInProgress THEN										// 	when Status has been changed within the block
	CASE CurrentMove.MoveType OF
		MoveTypeServo.Continuous :
				MCMoveVel (	Execute			:= FALSE,									//	reset MCMoves
							Axis			:= ioAxis);
		MoveTypeServo.LinearAbs :
				MCMoveAbs (	Execute			:= FALSE,
							Axis			:= ioAxis);
		MoveTypeServo.LinearRel :
				MCMoveRel (	Execute			:= FALSE,
							Axis			:= ioAxis);
	END_CASE		
	iCmd 						:= CmdServo.None;							//	clear command
END_IF
END_ACTION

ACTION Resetting:
MCReset( 	Execute				:= TRUE,										//	call fb to Reset axis
			Axis				:= ioAxis);										//
			
IF 	MCReset.Done THEN															//	if fb is Done (command successful)
	IF ioAxis.Status.Disabled THEN												//	check whether axis status is Disabled
		oState					:= StateServo.Disabled;							//	change status to Disabled
	ELSIF ioAxis.Status.StandStill THEN											//	or else if axis status is Standstill	
		oState					:= StateServo.Enabled;							//	change status to Enabled
	ELSIF ioAxis.Status.Error THEN												//	or else if axis status is Error
		oState					:= StateServo.Error;								//	change status to Error
	END_IF																		//
	MCReset( 	Execute			:= FALSE,										//	call Reset fb with Execute = false
				Axis			:= ioAxis);
ELSIF MCReset.Error THEN														//	if fb has an Error (command failed)
	oCmdFailed					:= TRUE;
	IF iCmdRetry THEN														//	command retry
		MCReset( 	Execute		:= FALSE,										//	call Reset fb with Execute = false
					Axis		:= ioAxis);										//	Reset fb will get retriggered on the next scan
		oCmdFailed				:= FALSE;
		iCmdRetry				:= FALSE;
	ELSIF iCmdAbort THEN													//	command abort
		MCReset( 	Execute		:= FALSE,										//	call Reset fb with Execute = false
					Axis		:= ioAxis);
		oState					:= PrevStatus;									//	change status back to Error
		oCmdFailed				:= FALSE;
		iCmdAbort				:= FALSE;
	END_IF
END_IF
END_ACTION

ACTION Stopped:
CASE iCmd OF
	CmdServo.Disable:																		//	accept the Disable command
					oState 								:= StateServo.Disabling;			//	change status to Disabling
					iCmd 								:= CmdServo.None;					//	clear command
	CmdServo.Home:																			//	accept the Disable command
					oState 								:= StateServo.Homing;				//	change status to Homing
					iCmd 								:= CmdServo.None;					//	clear command
	CmdServo.StartMove:																		//	accept the StartMove command
					ioMoves[iMoveIndex].Permissive();										//	check permissive
					IF NOT ioMoves[iMoveIndex].Permissive.Q THEN
						sMoveNotPermitted				:= TRUE;
						oCmdFailed						:= TRUE;
					ELSE
						sMoveNotPermitted				:= FALSE;
					END_IF
					
					MCMoveParametersCheck(	iMoveIndex 	:= iMoveIndex,						//	check parameters
											ioMoves 	:= ioMoves, 
											ioAxis 		:= ioAxis);
					IF NOT MCMoveParametersCheck.oValid THEN
						sMoveInvalid					:= TRUE;
						oCmdFailed						:= TRUE;
					ELSE
						sMoveInvalid					:= FALSE;
					END_IF
							
					IF  ioMoves[iMoveIndex].Permissive.Q AND MCMoveParametersCheck.oValid AND NOT oCmdFailed THEN
						CurrentMove 					:= ioMoves[iMoveIndex];
						oState 							:= StateServo.MoveInProgress;
						iCmd 							:= CmdServo.None;					//	clear command
					END_IF
					
					IF oCmdFailed AND iCmdRetry THEN
						oCmdFailed						:= FALSE;
						iCmdRetry						:= FALSE;
					ELSIF oCmdFailed AND iCmdAbort THEN
						oCmdFailed						:= FALSE;
						sMoveNotPermitted				:= FALSE;
						sMoveInvalid					:= FALSE;	
						iCmd	 						:= CmdServo.None;					//	clear command
						iCmdAbort						:= FALSE;
					END_IF															
	CmdServo.Jog:																			//	accept the Jog command
					oState 								:= StateServo.Jogging;				//	change status to Jogging
					iCmd 								:= CmdServo.None;					//	clear command
END_CASE

IF ioAxis.Status.Error THEN
	oState												:= StateServo.Error;
ELSIF ioAxis.status.Disabled THEN
	oState												:= StateServo.Disabled;
END_IF
END_ACTION

ACTION Stopping:
MCHalt(		Execute				:= TRUE,										//	call fb to Halt axis
			Axis				:= ioAxis);
IF 	MCHalt.Done AND ioaxis.Status.StandStill THEN								//	check for fb Done and axis status successfully changed to Standstill
	IF ioAxis.Status.Homed THEN													//	if axis has been homed
		oState 				:= StateServo.Stopped;							//	change status to Stopped
	ELSE																		//	if axis has not been homed (possible when jogging before homing)
		oState					:= StateServo.Enabled;							//	chagne status to Enabled
	END_IF
ELSIF MCHalt.Error THEN
	oCmdFailed				:= TRUE;
	IF iCmdRetry THEN														//	command retry
		MCHalt( 	Execute		:= FALSE,										//	call Halt fb with Execute = false
					Axis		:= ioAxis);										//	Home fb will get retriggered on the next scan
		oCmdFailed			:= FALSE;
		iCmdRetry			:= FALSE;
	ELSIF iCmdAbort THEN													//	command abort
		oState					:= PrevStatus;									//	change status back to previous
		oCmdFailed			:= FALSE;
		iCmdAbort			:= FALSE;
	END_IF
END_IF

IF 	iCmd = CmdServo.Disable THEN											//	accept the Disable command
	oState 					:= StateServo.Disabling;							//	change status to Disabling
END_IF

IF ioAxis.Status.Error THEN
	oState						:= StateServo.Error;
END_IF

IF oState <> StateServo.Stopping THEN											//	when Status has been changed within the block
	MCHalt( 	Execute			:= FALSE,										//	call Halt fb with Execute = false
				Axis			:= ioAxis);
	iCmd					:= CmdServo.None;								//	clear command
END_IF
END_ACTION

END_FUNCTION_BLOCK

// Instructions/MC_MoveParametersCheck
FUNCTION_BLOCK MC_MoveParametersCheck
VAR_INPUT
	iMoveIndex : INT;
END_VAR

VAR_OUTPUT
	oValid : BOOL;
END_VAR

VAR_IN_OUT
	ioAxis		: Axis_Ref;
	ioMoves 	: ARRAY [1..100] OF ServoMove;
END_VAR

VAR
	MCReadMaxVelocity		 	: MC_ReadParameter;
	MCReadMaxAccel				: MC_ReadParameter;
	MCReadMaxDecel				: MC_ReadParameter;
	MCReadMaxJerk				: MC_ReadParameter;
	MaxVelocity			: LREAL;
	MaxAccel			: LREAL;
	MaxDecel			: LREAL;
	MaxJerk				: LREAL;
END_VAR

MCReadMaxVelocity 	(	Enable 	:= TRUE,
						Axis	:= ioAxis,
						ParameterNumber := MC_AxisParameter.AxisMaxVelocity,
						ReadMode := E_ReadMode.READMODE_CYCLIC);

MCReadMaxAccel		(	Enable 	:= TRUE,
						Axis	:= ioAxis,
						ParameterNumber := MC_AxisParameter.AxisMaximumAcceleration,
						ReadMode := E_ReadMode.READMODE_CYCLIC);

MCReadMaxDecel		(	Enable 	:= TRUE,
						Axis	:= ioAxis,
						ParameterNumber := MC_AxisParameter.AxisMaximumDeceleration,
						ReadMode := E_ReadMode.READMODE_CYCLIC);

MCReadMaxJerk		(	Enable 	:= TRUE,
						Axis	:= ioAxis,
						ParameterNumber := MC_AxisParameter.MaxJerk,
						ReadMode := E_ReadMode.READMODE_CYCLIC);


MaxVelocity		:= MCReadMaxVelocity.Value;
MaxAccel		:= MCReadMaxAccel.Value;
MaxDecel		:= MCReadMaxDecel.Value;
MaxJerk			:= MCReadMaxJerk.Value;

IF 		ioMoves[iMoveIndex].Velocity > 0 AND ioMoves[iMoveIndex].Velocity < MaxVelocity AND 
		ioMoves[iMoveIndex].Accel > 0 AND ioMoves[iMoveIndex].Accel < MaxAccel AND 
		ioMoves[iMoveIndex].Decel > 0 AND ioMoves[iMoveIndex].Decel < MaxDecel AND
		ioMoves[iMoveIndex].Jerk >0 AND ioMoves[iMoveIndex].Jerk < MaxJerk AND
		ioMoves[iMoveIndex].MoveType <> MoveTypeServo.None THEN
					
	oValid := TRUE;
ELSE
	oValid := FALSE;	
END_IF

END_FUNCTION_BLOCK

// Instructions/eOR
FUNCTION_BLOCK eOR
VAR_INPUT
	IN1 : BOOL;
	IN2 : BOOL;
	IN3 : BOOL;
	IN4 : BOOL;
	IN5 : BOOL;
	IN6	: BOOL;
	IN7	: BOOL;
	IN8 : BOOL;
	IN9	: BOOL;
	IN10 : BOOL;

	Initialize : BOOL := TRUE;	
END_VAR

VAR_OUTPUT
	Q : BOOL;
END_VAR

VAR
	Input : ARRAY [1..10] OF eInput;	
	n : INT;
END_VAR

IF Initialize THEN
	IN1 := NOT Input[1].cActiveState;
	IN2 := NOT Input[2].cActiveState;
	IN3 := NOT Input[3].cActiveState;
	IN4 := NOT Input[4].cActiveState;
	IN5 := NOT Input[5].cActiveState;
	IN6 := NOT Input[6].cActiveState;
	IN7 := NOT Input[7].cActiveState;
	IN8 := NOT Input[8].cActiveState;
	IN9 := NOT Input[9].cActiveState;
	IN10 := NOT Input[10].cActiveState;	
END_IF

Input[1].iState := IN1;
Input[2].iState := IN2;
Input[3].iState := IN3;
Input[4].iState := IN4;
Input[5].iState := IN5;
Input[6].iState := IN6;
Input[7].iState := IN7;
Input[8].iState := IN8;
Input[9].iState := IN9;
Input[10].iState := IN10;


FOR n := 1 TO 10 BY 1 DO

		IF Input[n].iForceActive AND NOT Input[n].iForceInactive THEN
			Input[n].oActive := TRUE;
		ELSIF Input[n].iForceInactive AND NOT Input[n].iForceActive THEN
			Input[n].oActive := FALSE;
		ELSIF Input[n].cActiveState = Input[n].iState THEN
			Input[n].oActive := TRUE;
		ELSIF Input[n].cActiveState <> Input[n].iState THEN
			Input[n].oActive := FALSE;
		END_IF

END_FOR	

IF NOT Initialize THEN
Q := 	Input[1].oActive OR 
		Input[2].oActive OR 
		Input[3].oActive OR 
		Input[4].oActive OR 
		Input[5].oActive OR
		Input[6].oActive OR 
		Input[7].oActive OR 
		Input[8].oActive OR 
		Input[9].oActive OR 
		Input[10].oActive;
END_IF

Initialize := FALSE;

END_FUNCTION_BLOCK

// Instructions/StateManager
FUNCTION_BLOCK StateManager

VAR_INPUT
	iCmd 				: Cmd;
	iCmdRetry			: BOOL;
	iCmdAbort			: BOOL;
	iStartPermissives 	: eAND;
	iRunInterlocks 		: eAND;
	iSeqComplete 		: BOOL;
	iSeqFault			: BOOL;
END_VAR

VAR_INPUT PERSISTENT
	cAutoStart			: BOOL;
END_VAR

VAR_OUTPUT
	oState 				: State;
	oCmdFailed			: BOOL;
	sReadyToStart 		: BOOL;
	sCurrentRunTime 	: REAL;
	sPrevRunTime 		: REAL;
END_VAR

VAR_TEMP
	tmpRunTimer			: TIME;
END_VAR

VAR

END_VAR

iStartPermissives();
iRunInterlocks();

CASE oState OF
	State.Aborting:
						IF iSeqComplete THEN
							oState 				:= State.Aborted;
							iSeqComplete 		:= FALSE;
						ELSIF iSeqFault THEN
							oCmdFailed			:= TRUE;
						END_IF	
	
	State.Aborted : 	
						IF iCmd = Cmd.Reset THEN
							oState 				:= State.Resetting;
							iCmd				:= Cmd.None;
						END_IF
	
	State.Resetting : 	
						IF iSeqComplete THEN
							oState 				:= State.Stopped;
							iSeqComplete 		:= FALSE;
						ELSIF iSeqFault THEN
							oCmdFailed			:= TRUE;
						END_IF
						
						IF iCmd = Cmd.Abort THEN
							oState 				:= State.Aborting;
							iCmd				:= Cmd.None;
						END_IF
					
	State.Stopped :		
						IF cAutoStart AND iStartPermissives.Q AND iRunInterlocks.Q THEN
									oState 		:= State.Starting;
						END_IF
						
						CASE iCmd OF
							Cmd.Start:
								IF iStartPermissives.Q AND iRunInterlocks.Q AND NOT oCmdFailed THEN
									oState 		:= State.Starting;
									iCmd		:= Cmd.None;
								ELSE
									oCmdFailed	:= TRUE;
								END_IF
													
							Cmd.Abort:
									oState 		:= State.Aborting;
									iCmd		:= Cmd.None;
						END_CASE

	State.Starting :	
						IF iSeqComplete THEN
							oState 				:= State.Running;
							iSeqComplete 		:= FALSE;
						ELSIF iSeqFault THEN
							oCmdFailed			:= TRUE;
						END_IF
						
						CASE iCmd OF
							Cmd.Stop:
									oState 		:= State.Stopping;
									iCmd		:= Cmd.None;
							Cmd.Abort:
									oState 		:= State.Aborting;
									iCmd		:= Cmd.None;
						END_CASE

	State.Running :		
						IF iSeqComplete THEN
							oState 				:= State.Stopping;
							iSeqComplete 		:= FALSE;
						ELSIF NOT iRunInterlocks.Q THEN
									oState 		:= State.Pausing;
						END_IF
						
						CASE iCmd OF
							Cmd.Pause:
									oState 		:= State.Pausing;
									iCmd		:= Cmd.None;
							Cmd.Stop:
									oState 		:= State.Stopping;
									iCmd		:= Cmd.None;
							Cmd.Abort:
									oState 		:= State.Aborting;
									iCmd		:= Cmd.None;
						END_CASE	
						
	State.Pausing :
						IF iSeqComplete THEN
							oState 				:= State.Paused;
							iSeqComplete 		:= FALSE;
						END_IF
						
						CASE iCmd OF
							Cmd.Stop:
									oState 		:= State.Stopping;
									iCmd		:= Cmd.None;
							Cmd.Abort:
									oState 		:= State.Aborting;
									iCmd		:= Cmd.None;
						END_CASE
						
	State.Paused :
	
						CASE iCmd OF
							Cmd.Stop:
									oState 		:= State.Stopping;
									iCmd		:= Cmd.None;
							Cmd.Abort:
									oState 		:= State.Aborting;
									iCmd		:= Cmd.None;
						END_CASE
	
END_CASE

END_FUNCTION_BLOCK

// Instructions/Step
FUNCTION_BLOCK Step
VAR_INPUT
	iFaultCondition	: BOOL;
	iComplete		: BOOL;
	iRetry			: BOOL;
END_VAR

VAR_INPUT PERSISTENT
	cThisStep		: INT;
	cNextStep		: INT;
	cRecoveryStep	: INT;
	cTimeoutPreset	: TIME;
	cDescription	: STRING;
END_VAR

VAR_OUTPUT
	sActive			: BOOL;
	sFaulted		: BOOL;
	sTimedout		: BOOL;
	sComplete		: BOOL;
END_VAR

VAR_IN_OUT
	ioActiveStep	: INT;
END_VAR

VAR
	Status			: StatusStep;	
	ActiveTime		: TON;
END_VAR

ActiveTime.PT := cTimeoutPreset;

CASE Status OF
	StatusStep.Inactive:
							IF ioActiveStep = cThisStep THEN
								Status 			:= StatusStep.Active;
							END_IF
	StatusStep.Active:
							ActiveTime.IN 		:= TRUE;
							
							IF ActiveTime.Q THEN
								Status 			:= StatusStep.TimedOut;
								ActiveTime.IN 	:= FALSE;
							END_IF
							
							IF iFaultCondition THEN
								Status			:= StatusStep.Faulted;
							END_IF
							
							IF iComplete THEN
								Status			:= StatusStep.Complete;
							END_IF
	StatusStep.Faulted:
							IF iRetry THEN
								IF iFaultCondition = FALSE THEN
									Status			:= StatusStep.Active;
								ELSIF cRecoveryStep <> 0 THEN
									ioActiveStep := cRecoveryStep;
								END_IF
							END_IF
	StatusStep.TimedOut:
							IF iRetry THEN
								Status			:= StatusStep.Active;
							END_IF
	StatusStep.Complete:
							ioActiveStep := cNextStep;

END_CASE

END_FUNCTION_BLOCK
